{attribute 'qualified_only'}
VAR_GLOBAL
	Start					: BOOL;
	ReStart					: BOOL;
	Stop					: BOOL;
	Resume					: BOOL;
	ResetXTS_Error			: BOOL;
	dsMoverControlFlags		: MoverControlFlags;
	ShuttleMover			: BOOL;
	MachineState			: STRING;
	AutoMode				: BOOL;
	
	//Linked to SAFETY Alias
	LockDoors		AT %Q*	: BOOL;		
	
END_VAR

(* stored: Version 1.1.0.1, ProductVersion 3.1.4026.8
   GVL HMI: Id {74764eea-f9f1-0a62-209b-313e6c5f9e7d} *)
